// TIA Portal V16 export
// export: Created 2021-11-12T13:33:01.2606395Z, ExportSetting WithDefaults, DisplayName Totally Integrated Automation Portal, DisplayVersion V16 Update 3, DisplayName TIA Portal Version Control Interface, DisplayVersion V16 Update 2, DisplayName TIA Portal Openness, DisplayVersion V16 Update 3, DisplayName SINAMICS Startdrive Advanced, DisplayVersion V16 Update 5, DisplayName SINAMICS Startdrive G130, G150, S120, S150, SINAMICS MV, S210, DisplayVersion V16 Update 5, DisplayName SINAMICS Startdrive G110M, G120, G120C, G120D, G120P, G115D, DisplayVersion V16 Update 5, DisplayName STEP 7 Professional, DisplayVersion V16 Update 3, DisplayName STEP 7 Safety, DisplayVersion V16, DisplayName WinCC UA Professional, DisplayVersion V16 Update 3
DATA_BLOCK "STATUS_420"   // DB112
{ S7_Optimized_Access := 'TRUE' }
VERSION : 0.1
// stored: AutoNumber true, DBAccessibleFromOPCUA true, IsOnlyStoredInLoadMemory false, IsRetainMemResEnabled false, IsWriteProtectedInAS false, MemoryReserve 100
   VAR
      xxxxx___BinarySensors___xxxxx_1 : Byte;
      "EQ01-BL01" : Bool;   // Sensor for min surface (LSL1442) / Hladina min (LSL1442)
      "EQ01-BL02" : Bool;   // Sensor for max surface (LSH1443) / Hladina max (LSH1443)
      "EQ01-MA02_20" : Bool := FALSE;   // Valve (A1418) - closed
      "EQ01-MA02_24" : Bool := FALSE;   // Valve (A1418) - opened
      "EQ01-MA03_20" : Bool := FALSE;   // Valve (A1415) - closed
      "EQ01-MA03_24" : Bool := FALSE;   // Valve (A1415) - opened
      "EQ01-MA04_20" : Bool;   // Valve (A1412) - closed
      "EQ01-MA04_24" : Bool;   // Valve (A1412) - opened
      xxxxx___BinaryOthers___xxxxx_1 : Byte;
      "UC10-FC21_14" : Bool;   // 230V Hardening tube / 230V Zachlazovací nádrž
      "UC11-FC01_14" : Bool;   // 400V Pump of circulation P32 OK / 400V Čerpadlo cirkulace P32 OK
      DrainMode : Bool;   // Drain tank
      xxxxx___AnalogueSensors___xxxxx_1 : Byte;
      "EQ01-BT01" : Struct   // Temperature measurment (TIC 1425) / Měření teploty (TIC 1425)
         Main : "UDT_Status_main";
         Specific { S7_SetPoint := 'True'} : "UDT_CH_AI_Status_specific";
         Error { S7_SetPoint := 'True'} : "UDT_Error01";
      END_STRUCT;
      "EQ01-BP01" : Struct   // Tenzometric sond for measure surface (LIC 1431) / Tenzometrická sonda pro měření hladiny(LIC 1431)
         Main : "UDT_Status_main";
         Specific { S7_SetPoint := 'True'} : "UDT_CH_AI_Status_specific";
         Error { S7_SetPoint := 'True'} : "UDT_Error01";
      END_STRUCT;
      "EQ01-MA03_81" : Struct   // Valve analog indicator A 1415 Closed - opened / Meření ventilu A 1415 Zavřeno - otevřeno
         Main : "UDT_Status_main";
         Specific { S7_SetPoint := 'True'} : "UDT_CH_AI_Status_specific";
         Error { S7_SetPoint := 'True'} : "UDT_Error01";
      END_STRUCT;
      xxxxx___Drives___xxxxx_1 : Byte;
      "EQ01-MA01" : Struct   // Pump of circulation (P32) / Čerpadlo cirkulace (P32)
         Main : "UDT_Status_main";
         Specific : "UDT_Drive1_Status_specific";
         Error : "UDT_Error01";
      END_STRUCT;
      "EQ01-MA02" : Struct   // Valve with servomotor (A1418) / Ventil se servopohonem (A1418)
         Main { S7_SetPoint := 'True'} : "UDT_Status_main";
         Specific { S7_SetPoint := 'True'} : "UDT_Valve2WB_Status_specific";
         Error { S7_SetPoint := 'True'} : "UDT_Error01";
      END_STRUCT;
      "EQ01-MA03" : Struct   // Valve with servomotor (A1415) / Ventil se servopohonem (A1415)
         Main { S7_SetPoint := 'True'} : "UDT_Status_main";
         Specific { S7_SetPoint := 'True'} : "UDT_Valve2WB_Status_specific";
         Error { S7_SetPoint := 'True'} : "UDT_Error01";
      END_STRUCT;
      "EQ01-MA04" : Struct   // Valve with servomotor (A1412) / Ventil se servopohonem (A1412)
         Main { S7_SetPoint := 'True'} : "UDT_Status_main";
         Specific { S7_SetPoint := 'True'} : "UDT_Valve2WB_Status_specific";
         Error { S7_SetPoint := 'True'} : "UDT_Error01";
      END_STRUCT;
      "UC11-TA01" : Struct   // Frequence changer ( pro P32) / Frekvenční měnič ( pro P32)
         Main : "UDT_Status_main";
         Specific : "UDT_SINAMICS_G120_Status_specific";
         Error : "UDT_Error02";
      END_STRUCT;
      xxxxx___Alarms___xxxxx : Byte;
      ES : Struct   // E-stop
         Main { S7_SetPoint := 'True'} : "UDT_Status_main";
         Specific { S7_SetPoint := 'True'} : "UDT_DI_Mon_Status_specific";
         Error { S7_SetPoint := 'True'} : "UDT_Error01";
      END_STRUCT;
      KF31 : Struct   // Module KF31 / Modul KF31
         Main { S7_SetPoint := 'True'} : "UDT_Status_main";
         Specific { S7_SetPoint := 'True'} : "UDT_DI_Mon_Status_specific";
         Error { S7_SetPoint := 'True'} : "UDT_Error01";
      END_STRUCT;
      EQ01_BL01 : Struct   // Sensor Max level active and sensor Min level / Aktivní senzor vysoké hladiny a neaktivní senzor nízké hladiny.
         Main : "UDT_Status_main";
         Specific { S7_SetPoint := 'True'} : "UDT_DI_Mon_Status_specific";
         Error { S7_SetPoint := 'True'} : "UDT_Error01";
      END_STRUCT;
      EQ01_BL02 : Struct   // Sensor Min level active and analog level sensor under 10% / Senzor minimální hladiny aktivní a analogový senzor pod 10%.
         Main : "UDT_Status_main";
         Specific { S7_SetPoint := 'True'} : "UDT_DI_Mon_Status_specific";
         Error { S7_SetPoint := 'True'} : "UDT_Error01";
      END_STRUCT;
      EQ01_BP01 : Struct   // Analog level sensor over 40% and sensor min level not active / Vodní hladina nad 40% a senzor minimální hladiny neaktivní.
         Main : "UDT_Status_main";
         Specific { S7_SetPoint := 'True'} : "UDT_DI_Mon_Status_specific";
         Error { S7_SetPoint := 'True'} : "UDT_Error01";
      END_STRUCT;
      Water_temp_high : Struct   // Water temperature high / Teplota vody nad vrchní tolerancí.
         Main : "UDT_Status_main";
         Specific { S7_SetPoint := 'True'} : "UDT_DI_Mon_Status_specific";
         Error { S7_SetPoint := 'True'} : "UDT_Error01";
      END_STRUCT;
      Water_temp_low : Struct   // Water temperature low / Teplota vody pod spodnou tolerancí.
         Main : "UDT_Status_main";
         Specific { S7_SetPoint := 'True'} : "UDT_DI_Mon_Status_specific";
         Error { S7_SetPoint := 'True'} : "UDT_Error01";
      END_STRUCT;
      Water_level_high : Struct   // Water level high / Vysoká hladina vody.
         Main : "UDT_Status_main";
         Specific { S7_SetPoint := 'True'} : "UDT_DI_Mon_Status_specific";
         Error { S7_SetPoint := 'True'} : "UDT_Error01";
      END_STRUCT;
      Level_NOK : Struct   // BSN4 tacts and water level NOK / BSN4 taktuje a hladina vody je NOK
         Main : "UDT_Status_main";
         Specific { S7_SetPoint := 'True'} : "UDT_DI_Mon_Status_specific";
         Error { S7_SetPoint := 'True'} : "UDT_Error01";
      END_STRUCT;
      EQ01_MA04 : Struct   // Filling and no water level change / Chyba napouštení, hladina nezměnena
         Main : "UDT_Status_main";
         Specific { S7_SetPoint := 'True'} : "UDT_DI_Mon_Status_specific";
         Error { S7_SetPoint := 'True'} : "UDT_Error01";
      END_STRUCT;
      EQ01_MA02 : Struct   // Drain and no water level change / Chyba vypouštení, hladina nezměnena
         Main : "UDT_Status_main";
         Specific { S7_SetPoint := 'True'} : "UDT_DI_Mon_Status_specific";
         Error { S7_SetPoint := 'True'} : "UDT_Error01";
      END_STRUCT;
   END_VAR
BEGIN
END_DATA_BLOCK
